Fanuc KAREL source: kt00521.compact.KL

PROGRAM KT00521
%STACKSIZE=65535
%PRIORITY=65535
%NOLOCKGROUP
VAR
P1 : XYZWPREXT
P2 : XYZWPR
OUT : XYZWPREXT
BEGIN
P1.X=1.0
P2.Y=2.0
OUT=P1 : P2
END KT00521
